// Mitsubishi GX Works2 project: Fx1s-Button-Light   PLC: FX1S

PROGRAM MAIN
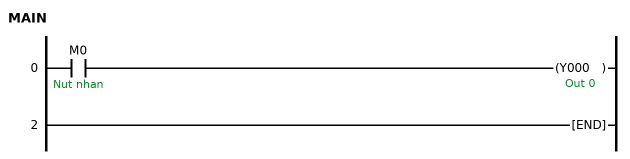
0     LD      M0  ; Nut nhan
      OUT     Y000  ; Out 0
2     END
END_PROGRAM
